TYPE MaterialXMapping :
STRUCT
	{attribute 'OPC.UA.DA.Description' := 'Type ID of material'}
	MaterialTypeID				: STRING(30);

	{attribute 'OPC.UA.DA.Description' := 'Location material is configured on'}
	Location					: UINT;

END_STRUCT
END_TYPE

(* stored: Version 1.1.0.1, ProductVersion 3.1.4024.5
   DUT MaterialXMapping: Id {89746586-44f3-4e4a-bd15-5d415c421946} *)
